FUNCTION_BLOCK MathTest EXTENDS TcUnit.FB_TestSuite

Test_Cbrt();
Test_LrealFromBits();
Test_Ceil();
Test_Fmod();
Test_Clamp();

METHOD Test_Cbrt
VAR
  actual : LREAL;
END_VAR
TEST('Cbrt');

actual := Struckig.Cbrt(8);
AssertEquals_LREAL(2, actual, 1E-20, message:='');

actual := Struckig.Cbrt(-8);
AssertEquals_LREAL(-2, actual, 1E-20, message:='');

actual := Struckig.Cbrt(5E-18);
AssertEquals_LREAL(1.70997594667669698E-6, actual, 1E-18, message:='');

actual := Struckig.Cbrt(0.5);
AssertEquals_LREAL(0.793700525984099737, actual, 1E-18, message:='');

actual := Struckig.Cbrt(3.5353238602192074E-08);
AssertEquals_LREAL(0.0032820339420509366, actual, 1E-18, message:='');

TEST_FINISHED();
END_METHOD

METHOD Test_Ceil
VAR
  actual : LREAL;
END_VAR
TEST('Ceil');

actual := Struckig.Ceil(8.1);
AssertEquals_LREAL(9, actual, 1E-20, message:='');

actual := Struckig.Ceil(-8.1);
AssertEquals_LREAL(-8, actual, 1E-20, message:='');

actual := Struckig.Ceil(0);
AssertEquals_LREAL(0, actual, 1E-20, message:='');

actual := Struckig.Ceil(0.1);
AssertEquals_LREAL(1, actual, 1E-20, message:='');

actual := Struckig.Ceil(-0.1);
AssertEquals_LREAL(0, actual, 1E-20, message:='');

TEST_FINISHED();
END_METHOD

METHOD Test_Clamp
VAR
  actual : LREAL;
END_VAR
TEST('Clamp');

actual := Struckig.Clamp(-1, 0, 1);
AssertEquals_LREAL(0, actual, 1E-20, message:='');

actual := Struckig.Clamp(-1, -2, 1);
AssertEquals_LREAL(-1, actual, 1E-20, message:='');

actual := Struckig.Clamp(2, 0, 1);
AssertEquals_LREAL(1, actual, 1E-20, message:='');

TEST_FINISHED();
END_METHOD

METHOD Test_Fmod
VAR
  actual : LREAL;
END_VAR
TEST('Cbrt');

actual := Struckig.Fmod(5, 1);
AssertEquals_LREAL(0, actual, 1E-20, message:='');

actual := Struckig.Fmod(5, 2);
AssertEquals_LREAL(1, actual, 1E-20, message:='');

actual := Struckig.Fmod(5, 3);
AssertEquals_LREAL(2, actual, 1E-20, message:='');

actual := Struckig.Fmod(5, 4);
AssertEquals_LREAL(1, actual, 1E-20, message:='');

actual := Struckig.Fmod(5, 5);
AssertEquals_LREAL(0, actual, 1E-20, message:='');

actual := Struckig.Fmod(5, 6);
AssertEquals_LREAL(5, actual, 1E-20, message:='');

actual := Struckig.Fmod(5, 7);
AssertEquals_LREAL(5, actual, 1E-20, message:='');

actual := Struckig.Fmod(5, 8);
AssertEquals_LREAL(5, actual, 1E-20, message:='');

actual := Struckig.Fmod(123.123, 0.121);
AssertEquals_LREAL(0.066, actual, 1E-20, message:='');

TEST_FINISHED();
END_METHOD

METHOD Test_LrealFromBits
VAR
  actual : LREAL;
END_VAR
TEST('LrealFromBits');

actual := Struckig.LrealFromBits(1);
AssertEquals_LREAL(4.94065645841247E-324, actual, 0, message:=''); // Epsilon

actual := Struckig.LrealFromBits(0);
AssertEquals_LREAL(0, actual, 0, message:='');

TEST_FINISHED();
END_METHOD

END_FUNCTION_BLOCK

(* stored: Version 1.1.0.1
   POU MathTest: Id {db8e1fc4-323a-4e57-889c-7de3202bf79d}, SpecialFunc None
   Method Test_Cbrt: Id {fb4f66a2-1f91-4a1e-b1d2-83e0fdba8205}
   Method Test_Ceil: Id {9fd4e64d-fdec-4ee2-a367-51305cf91684}
   Method Test_Clamp: Id {0b9dcc11-6cdc-4240-8723-22092748cb1a}
   Method Test_Fmod: Id {2d283eca-8afb-4973-8ca2-2aedc13f57fa}
   Method Test_LrealFromBits: Id {65953fc4-9b2c-43c4-9a3b-522ec2add867} *)
